TYPE "txRecordReadSto"
TITLE = {"version":"v1.0","author":"cyanezf","family":"core/fieldbus/lldx","status":"current","deprecatedBy": null,"dependencies":[]}

//(*--
//# Documentation
//## Log
//| version | date | author | description |
//|:-------:|:----:|:------:|:------------|
//| v1.0 | 2022-10-12 | cyanezf | First version |
//
//## Description
//TX record read storage
//--*)

   STRUCT
      ackCounter : Byte;   // El receptor confirma la lectura del juego de datos escribiendo el valor de la entrada cycle_counter en la salida ack_counter. A continuación, el juego de datos se borra de la memoria de respaldo
   END_STRUCT;

END_TYPE

